FUNCTION_BLOCK FB_BacklashCompensationNC_TestDouble IMPLEMENTS I_BacklashCompensation
VAR
    bError : BOOL;
    nErrorID : UDINT := 21000;
END_VAR

{warning 'Add method implementation '}
METHOD BacklashCompensation
VAR_INPUT
    Enable	: BOOL := FALSE;
    RampVelo	: LREAL;
END_VAR
END_METHOD

{warning 'Add method implementation '}
METHOD BacklashCompensationTest
VAR_INPUT
    UserEnable	: BOOL;
    Compensation	: LREAL;
END_VAR
END_METHOD

{warning 'Add property implementation'}
PROPERTY Busy : BOOL
GET
END_GET
END_PROPERTY

{warning 'Add property implementation'}
PROPERTY CurrentBacklash : LREAL
GET
END_GET
END_PROPERTY

{warning 'Add property implementation'}
PROPERTY Enable : BOOL
SET
END_SET
END_PROPERTY

{warning 'Add property implementation'}
PROPERTY Error : BOOL
GET
Error := bError;
END_GET
SET
bError := Error;
END_SET
END_PROPERTY

{warning 'Add property implementation'}
PROPERTY ErrorID : UDINT
GET
ErrorId := nErrorID;
END_GET
SET
nErrorId := ErrorID;
END_SET
END_PROPERTY

{warning 'Add property implementation'}
PROPERTY Message : T_MAXSTRING
GET
END_GET
END_PROPERTY

{warning 'Add property implementation'}
PROPERTY Status : BOOL
GET
END_GET
END_PROPERTY

{warning 'Add property implementation'}
PROPERTY UserEnable : BOOL
SET
END_SET
END_PROPERTY

END_FUNCTION_BLOCK

(* stored: Version 1.1.0.1
   POU FB_BacklashCompensationNC_TestDouble: Id {c8ccd65b-c409-4be0-a30d-cd79c23753d7}, SpecialFunc None
   Method BacklashCompensation: Id {a8547e2a-8dbe-4226-b04b-f971f495e78e}
   Method BacklashCompensationTest: Id {8c3ba61d-867b-40b8-bc1e-997154128749}
   Property Busy: Id {9e505eab-e76e-489b-b78d-bdc22ecb670a}
   Get Get: Id {00ba005e-b995-4294-b9dd-7001e8477fe7}
   Property CurrentBacklash: Id {4eb4a049-4acb-4178-a1ce-5c2c00642f0f}
   Get Get: Id {7f63c098-d429-4bd1-9dd3-e3dddd4ff751}
   Property Enable: Id {778f6f4d-c5c8-4f60-99af-e407231d6461}
   Set Set: Id {c1b50366-cd8b-48c4-9098-17ac5eabbb08}
   Property Error: Id {b0357fa8-7313-4690-929f-eefb5e8d200b}
   Get Get: Id {a055e96b-5bda-47a1-8cb1-8a68eabd8397}
   Set Set: Id {a45ca64f-86f9-4112-bad3-4a23ea393471}
   Property ErrorID: Id {d318f7d1-5e87-4588-bcc8-6ddec58a65dc}
   Get Get: Id {a5a056ea-0c82-4e1b-a141-bbe694f0368d}
   Set Set: Id {dbfaad40-87ca-484b-8898-97ba4a3606a3}
   Property Message: Id {a848a9ed-5ad8-48c7-95f4-8f4ff86a5d1d}
   Get Get: Id {6f7a0cb6-f62c-45ea-bace-5bbf583e3c21}
   Property Status: Id {718cc66e-d592-4762-940b-2a3810dc2588}
   Get Get: Id {74616016-a8eb-43ec-b466-1ceb5c10a6f9}
   Property UserEnable: Id {62bd6129-2ad1-4d43-b147-27ce7bb1ac45}
   Set Set: Id {697e3ba8-382a-4f29-b2c3-b83c3718f3ed} *)
